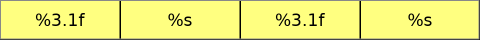
VISUALIZATION VISU_CONFIG_LIGNE_GAZ_SURV_MFC_MKS  // 480x40
VAR_IN_OUT
	m_Input_MASSFLOW:		BLOCK_MFC_MKS_NoCoE;
END_VAR
    Rectangle (0,0 120x40), "%3.1f", text variable: m_Input_MASSFLOW.VAR_ALM_SURV.OFFSET, input disabled if: NOT Global_Variables.PRG_USER.ACTU_USER.CONF_MACHINE
        OnMouseDown: write the text variable via Edit
    Rectangle (240,0 120x40), "%3.1f", text variable: m_Input_MASSFLOW.VAR_DEF_SURV.offset, input disabled if: NOT Global_Variables.PRG_USER.ACTU_USER.CONF_MACHINE
        OnMouseDown: write the text variable via VisuDialogs.Numpad
    Rectangle (120,0 120x40), "%s", text variable: m_Input_MASSFLOW.ALM_SURV.delay, input disabled if: NOT Global_Variables.PRG_USER.ACTU_USER.CONF_MACHINE
        OnMouseDown: write the text variable via VisuDialogs.Keypad
    Rectangle (360,0 120x40), "%s", text variable: m_Input_MASSFLOW.DEF_SURV.DELAY, input disabled if: NOT Global_Variables.PRG_USER.ACTU_USER.CONF_MACHINE
        OnMouseDown: write the text variable via VisuDialogs.Keypad
END_VISUALIZATION

// ---- Visualizations/Symbole/GAZ/VISU_CONFIG_REGUL_GAZ.TcVIS
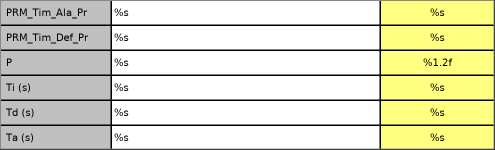
VISUALIZATION VISU_CONFIG_REGUL_GAZ  // 495x150
VAR_IN_OUT
	m_Input_REGULATION : BLOCK_REGUL_PR_GAZ;
END_VAR
    Rectangle (111,50 269x25), "%s", text list: 'TextList_Config_Gaz', text index: 31
    Rectangle (380,50 115x25), "%1.2f", text variable: m_Input_REGULATION.CONTROLEUR_GAZ.CONF_Kp, input disabled if: NOT Global_Variables.PRG_USER.ACTU_USER.CONF_MACHINE
        OnMouseDown: write the text variable via InputWithLimits, min 0
    Rectangle (0,50 111x25), "P", text variable: 1
    Rectangle (111,75 269x25), "%s", text list: 'TextList_Config_Gaz', text index: 32
    Rectangle (111,100 269x25), "%s", text list: 'TextList_Config_Gaz', text index: 33
    Rectangle (380,75 115x25), "%s", text variable: m_Input_REGULATION.CONTROLEUR_GAZ.CONF_Tn, input disabled if: NOT Global_Variables.PRG_USER.ACTU_USER.CONF_MACHINE
        OnMouseDown: write the text variable via InputWithLimits
    Rectangle (0,75 111x25), "Ti (s)", text variable: 1
    Rectangle (380,100 115x25), "%s", text variable: m_Input_REGULATION.CONTROLEUR_GAZ.CONF_Tv, input disabled if: NOT Global_Variables.PRG_USER.ACTU_USER.CONF_MACHINE
        OnMouseDown: write the text variable via InputWithLimits
    Rectangle (0,100 111x25), "Td (s)", text variable: 1
    Rectangle (111,125 269x25), "%s", text list: 'TextList_Config_Gaz', text index: 34
    Rectangle (380,125 115x25), "%s", text variable: m_Input_REGULATION.CONTROLEUR_GAZ.CONF_Td, input disabled if: NOT Global_Variables.PRG_USER.ACTU_USER.CONF_MACHINE
        OnMouseDown: write the text variable via InputWithLimits
    Rectangle (0,125 111x25), "Ta (s)", text variable: 1
    Rectangle (111,0 269x25), "%s", text list: 'TextList_Config_Gaz', text index: 29
    Rectangle (380,0 115x25), "%s", text variable: m_Input_REGULATION.PRM_Tim_Ala_Pr, input disabled if: NOT Global_Variables.PRG_USER.ACTU_USER.CONF_MACHINE
        OnMouseDown: write the text variable via InputWithLimits
    Rectangle (0,0 111x25), "PRM_Tim_Ala_Pr"
    Rectangle (111,25 269x25), "%s", text list: 'TextList_Config_Gaz', text index: 30
    Rectangle (380,25 115x25), "%s", text variable: m_Input_REGULATION.PRM_Tim_Def_Pr, input disabled if: NOT Global_Variables.PRG_USER.ACTU_USER.CONF_MACHINE
        OnMouseDown: write the text variable via InputWithLimits
    Rectangle (0,25 111x25), "PRM_Tim_Def_Pr"
END_VISUALIZATION

// ---- Visualizations/Symbole/GAZ/VISU_LIGNE_GAZ.TcVIS
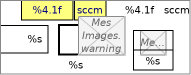
VISUALIZATION VISU_LIGNE_GAZ  // 191x75
VAR_IN_OUT
	m_Input_MACHINE:	BLOCK_MODE_MARCHE_V2_0;
	m_Input_MASSFLOW:	BLOCK_MFC_BROOKS_NoCoE;
	m_Input_LIGNE_GAZ:	BLOCK_LIGNE_GAZ;
END_VAR
    Frame (21,0 170x75)
        shows VISU_MFC_BROOKS(m_Input_MACHINE := m_Input_MACHINE, m_Input_MASSFLOW := m_Input_MASSFLOW, m_Input_LIGNE_GAZ := m_Input_LIGNE_GAZ)
    Frame (133,30 42x42)
        shows VISU_VANNE_2P_H_ACT2(m_Input_VANNE := m_Input_LIGNE_GAZ.VGI)
    Rectangle (0,25 48x28), "%s", text variable: m_Input_MASSFLOW.CONF_Util_Name
END_VISUALIZATION

// ---- Visualizations/Symbole/GAZ/VISU_LIGNE_GAZ_ANA.TcVIS
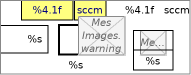
VISUALIZATION VISU_LIGNE_GAZ_ANA  // 191x75
VAR_IN_OUT
	m_Input_MACHINE:	BLOCK_MODE_MARCHE_V2_0;
	m_Input_MASSFLOW:	BLOCK_MFC_ANA2;
	m_Input_LIGNE_GAZ:	BLOCK_LIGNE_GAZ;		
END_VAR
    Frame (21,0 170x75)
        shows VISU_MFC_ANA(m_Input_MACHINE := m_Input_MACHINE, m_Input_MASSFLOW := m_Input_MASSFLOW, m_Input_LIGNE_GAZ := m_Input_LIGNE_GAZ)
    Frame (133,30 42x42)
        shows VISU_VANNE_2P_H_ACT2(m_Input_VANNE := m_Input_LIGNE_GAZ.VGI)
    Rectangle (0,25 48x28), "%s", text variable: m_Input_MASSFLOW.CONF_Util_Name
END_VISUALIZATION

// ---- Visualizations/Symbole/GAZ/VISU_LIGNE_GAZ_VGAUCHE.TcVIS
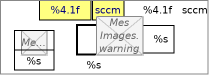
VISUALIZATION VISU_LIGNE_GAZ_VGAUCHE  // 209x75
VAR_IN_OUT
	m_Input_MACHINE:	BLOCK_MODE_MARCHE_V2_0;
	m_Input_MASSFLOW:	BLOCK_MFC_MKS_NoCoE;
	m_Input_LIGNE_GAZ:	BLOCK_LIGNE_GAZ;
END_VAR
    Frame (14,30 42x42)
        shows VISU_VANNE_2P_H_ACT2(m_Input_VANNE := m_Input_LIGNE_GAZ.VGI)
    Rectangle (126,25 48x28), "%s", text variable: m_Input_MASSFLOW.CONF_Util_Name
    Frame (39,0 170x75)
        shows VISU_MFC_MKS(m_Input_MACHINE := m_Input_MACHINE, m_Input_MASSFLOW := m_Input_MASSFLOW, m_Input_LIGNE_GAZ := m_Input_LIGNE_GAZ)
        p3089095539: m_Input_MACHINE
        p1532468285: m_Input_MASSFLOW
        p4266626122: m_Input_LIGNE_GAZ
END_VISUALIZATION

// ---- Visualizations/Symbole/GAZ/VISU_MFC_ANA.TcVIS
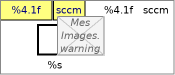
VISUALIZATION VISU_MFC_ANA  // 175x75
VAR_IN_OUT
	m_Input_MACHINE:	BLOCK_MODE_MARCHE_V2_0;
	m_Input_MASSFLOW:	BLOCK_MFC_ANA2;
	m_Input_LIGNE_GAZ:	BLOCK_LIGNE_GAZ;
END_VAR
    Rectangle (37,24 34x31)
    RoundedRectangle (0,0 52x20), "%4.1f", text variable: m_Input_MASSFLOW.PRM_Flow, invisible if: (m_Input_MACHINE.STATE_Manu) <> 0
    Rectangle (90,0 49x20), "%4.1f", text variable: m_Input_MASSFLOW.STATE_Flow
    RoundedRectangle (53,0 32x20), "sccm"
    Rectangle (140,0 35x20), "sccm"
    Rectangle (35,55 40x20), "%s", text variable: m_Input_MASSFLOW.MNEMO
    RoundedRectangle (0,0 52x20), "%4.1f", text variable: m_Input_LIGNE_GAZ.PRM_Flow, invisible if: NOT m_Input_MACHINE.STATE_Manu, input disabled if: NOT m_Input_MACHINE.STATE_Manu OR NOT PRG_User.ACTU_USER.MAINTENANCE
        OnMouseDown: write the text variable via VisuDialogs.Numpad, min 0, max m_Input_MASSFLOW.CONF_Util_Max_Flow
    Polyline (53,32)
    Polyline (61,39)
    Rectangle (55,39 16x18), "D"
    Image (57,16 47x39), invisible if: NOT m_Input_MASSFLOW.STATE_NOK, image: MesImages.warning
END_VISUALIZATION

// ---- Visualizations/Symbole/GAZ/VISU_MFC_BROOKS.TcVIS
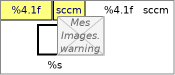
VISUALIZATION VISU_MFC_BROOKS  // 175x75
VAR_IN_OUT
	m_Input_MACHINE:	BLOCK_MODE_MARCHE_V2_0;
	m_Input_MASSFLOW:	BLOCK_MFC_BROOKS_NoCoE;
	m_Input_LIGNE_GAZ:	BLOCK_LIGNE_GAZ;
END_VAR
    Rectangle (37,24 34x31)
    RoundedRectangle (0,0 52x20), "%4.1f", text variable: m_Input_MASSFLOW.PRM_Flow, invisible if: NOT m_Input_MACHINE.STATE_Manu, input disabled if: NOT m_Input_MACHINE.STATE_Manu OR NOT PRG_User.ACTU_USER.MAINTENANCE
    Rectangle (90,0 49x20), "%4.1f", text variable: m_Input_MASSFLOW.STATE_Flow
    RoundedRectangle (53,0 32x20), "sccm"
    Rectangle (140,0 35x20), "sccm"
    Rectangle (35,55 40x20), "%s", text variable: m_Input_MASSFLOW.MNEMO
    RoundedRectangle (0,0 52x20), "%4.1f", text variable: m_Input_LIGNE_GAZ.PRM_Flow, invisible if: NOT m_Input_MACHINE.STATE_Manu, input disabled if: NOT m_Input_MACHINE.STATE_Manu OR NOT PRG_User.ACTU_USER.MAINTENANCE
        OnMouseDown: write the text variable via InputWithLimits, min 0, max m_Input_MASSFLOW.CONF_Util_Max_Flow
    Polyline (53,32)
    Polyline (61,39)
    Rectangle (55,39 16x18), "D"
    Image (57,16 47x39), invisible if: NOT m_Input_MASSFLOW.STATE_NOK, image: MesImages.warning
END_VISUALIZATION

// ---- Visualizations/Symbole/GAZ/VISU_MFC_MKS.TcVIS
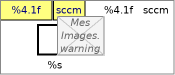
VISUALIZATION VISU_MFC_MKS  // 175x75
VAR_IN_OUT
	m_Input_MACHINE:	BLOCK_MODE_MARCHE_V2_0;
	m_Input_MASSFLOW:	BLOCK_MFC_MKS_NoCoE;
	m_Input_LIGNE_GAZ:	BLOCK_LIGNE_GAZ;
END_VAR
    Rectangle (37,24 34x31)
    RoundedRectangle (0,0 52x20), "%4.1f", text variable: m_Input_MASSFLOW.PRM_Flow, invisible if: (m_Input_MACHINE.STATE_Manu) <> 0
    Rectangle (90,0 49x20), "%4.1f", text variable: m_Input_MASSFLOW.STATE_Flow
    RoundedRectangle (53,0 32x20), "sccm"
    Rectangle (140,0 35x20), "sccm"
    Rectangle (35,55 40x20), "%s", text variable: m_Input_MASSFLOW.MNEMO
    RoundedRectangle (0,0 52x20), "%4.1f", text variable: m_Input_LIGNE_GAZ.PRM_Flow, invisible if: NOT m_Input_MACHINE.STATE_Manu, input disabled if: NOT m_Input_MACHINE.STATE_Manu OR NOT PRG_User.ACTU_USER.MAINTENANCE
        OnMouseDown: write the text variable via VisuDialogs.Numpad, min 0, max m_Input_MASSFLOW.CONF_Util_Max_Flow
    Polyline (53,32)
    Polyline (61,39)
    Rectangle (55,39 16x18), "D"
    Image (57,16 47x39), invisible if: NOT m_Input_MASSFLOW.STATE_NOK, image: MesImages.warning
END_VISUALIZATION

// ---- Visualizations/Symbole/IAD/VISU_MARK3_PLUS.TcVIS
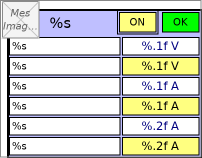
VISUALIZATION VISU_MARK3_PLUS  // 202x158
VAR_IN_OUT
	m_Input_IAD : BLOCK_MARK3_PLUS;
END_VAR
    Rectangle (7,9 195x149)
    Rectangle (162,12 37x20), "NOK", invisible if: (m_Input_IAD.IN_BUSSTAT) <> 0
    Rectangle (119,12 37x20), "OFF", invisible if: (m_Input_IAD.STATE_BEAM OR m_Input_IAD.STATE_BEAM_ON) <> 0
    Rectangle (162,12 37x20), "OK", invisible if: NOT m_Input_IAD.IN_BUSSTAT
    Rectangle (119,12 37x20), "ON", invisible if: NOT m_Input_IAD.STATE_BEAM AND NOT m_Input_IAD.STATE_BEAM_ON
    RoundedRectangle (9,37 111x18), "%s", text list: 'TextList_IAD', text index: 0
    RoundedRectangle (122,37 77x18), "%.1f V", text variable: m_Input_IAD.STATE_V_Anode
    RoundedRectangle (9,77 111x18), "%s", text list: 'TextList_IAD', text index: 1
    RoundedRectangle (122,77 77x18), "%.1f A", text variable: m_Input_IAD.STATE_I_Anode
    Rectangle (119,12 37x20), "ON", invisible if: (m_Input_IAD.STATE_BEAM_ON OR NOT m_Input_IAD.STATE_BEAM) <> 0
    Rectangle (7,12 107x22), "%s", text variable: m_Input_IAD.MNEMO
    Polyline (7,35)
    RoundedRectangle (9,57 111x18), "%s", invisible if: NOT Global_Variables.PRG_USER.ACTU_USER.MAINTENANCE OR NOT MACHINE.State_manu, text list: 'TextList_IAD', text index: 0
    RoundedRectangle (122,57 77x18), "%.1f V", text variable: m_Input_IAD.PRM_ANODE_VOLTAGE, invisible if: NOT Global_Variables.PRG_USER.ACTU_USER.MAINTENANCE OR NOT MACHINE.State_manu
        OnMouseDown: write the text variable via VisuDialogs.Numpad, min 0, max 300
    RoundedRectangle (9,97 111x18), "%s", invisible if: NOT Global_Variables.PRG_USER.ACTU_USER.MAINTENANCE OR NOT MACHINE.State_manu, text list: 'TextList_IAD', text index: 1
    RoundedRectangle (122,97 77x18), "%.1f A", text variable: m_Input_IAD.PRM_ANODE_CURRENT, invisible if: NOT Global_Variables.PRG_USER.ACTU_USER.MAINTENANCE OR NOT MACHINE.State_manu
        OnMouseDown: write the text variable via VisuDialogs.Numpad, min 0, max 15
    Rectangle (117,10 41x24), invisible if: NOT m_Input_IAD.BEAM.AUTOR_ON_IHM AND NOT m_Input_IAD.BEAM.AUTOR_OFF_IHM, input disabled if: ((NOT m_Input_IAD.BEAM.AUTOR_ON_IHM AND NOT m_Input_IAD.BEAM.AUTOR_OFF_IHM) OR NOT PRG_User.ACTU_USER.MAINTENANCE) <> 0
        OnMouseUp: execute { m_Input_IAD.BEAM.M_On:=(TRUE); }
    RoundedRectangle (9,117 111x18), "%s", text list: 'TextList_IAD', text index: 2
    RoundedRectangle (122,117 77x18), "%.2f A", text variable: m_Input_IAD.STATE_I_Neut
    RoundedRectangle (9,137 111x18), "%s", invisible if: NOT Global_Variables.PRG_USER.ACTU_USER.MAINTENANCE OR NOT MACHINE.State_manu, text list: 'TextList_IAD', text index: 2
    RoundedRectangle (122,137 77x18), "%.2f A", text variable: m_Input_IAD.PRM_NEUTRAL_CURRENT, invisible if: NOT Global_Variables.PRG_USER.ACTU_USER.MAINTENANCE OR NOT MACHINE.State_manu
        OnMouseDown: write the text variable via VisuDialogs.Numpad, min 0, max 1.86
    Image (2,1 37x37), invisible if: NOT m_Input_IAD.STATE_Nok, image: MesImages.warning
END_VISUALIZATION

// ---- Visualizations/Symbole/IAD/VISU_MARK3_PLUS_COTE.TcVIS
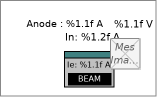
VISUALIZATION VISU_MARK3_PLUS_COTE  // 157x97
VAR_IN_OUT
	m_Input_IAD : BLOCK_MARK3_PLUS;
END_VAR
    Polygon (59,48), invisible if: NOT m_Input_IAD.STATE_BEAM_ON
    Polygon (91,50), invisible if: NOT m_Input_IAD.STATE_BEAM_ON
    Polygon (86,81)
    Rectangle (85,69 25x10), "ON"
    RoundedRectangle (64,51 50x36)
    Rectangle (64,51 50x7)
    RoundedRectangle (68,73 43x12), "BEAM", colour toggle: (m_Input_IAD.STATE_BEAM_ON) <> 0
    Rectangle (51,58 76x14), "Ie: %1.1f A", text variable: m_Input_IAD.STATE_I_Emi, invisible if: NOT m_Input_IAD.STATE_BEAM
    Rectangle (63,52 52x32), input disabled if: ((NOT m_Input_IAD.BEAM.AUTOR_ON_IHM AND NOT m_Input_IAD.BEAM.AUTOR_OFF_IHM) OR NOT PRG_User.ACTU_USER.MAINTENANCE) <> 0
        OnMouseUp: execute { m_Input_IAD.BEAM.M_On:=(TRUE); }
    RoundedRectangle (68,73 43x12), "BEAM", invisible if: (m_Input_IAD.STATE_BEAM_ON OR m_Input_IAD.STATE_BEAM) <> 0
    Rectangle (25,17 83x14), "Anode : %1.1f A", text variable: m_Input_IAD.STATE_I_Anode, invisible if: NOT m_Input_IAD.STATE_BEAM
    Rectangle (107,17 50x14), "%1.1f V", text variable: m_Input_IAD.STATE_V_Anode, invisible if: NOT m_Input_IAD.STATE_BEAM
    Rectangle (60,30 62x14), "In: %1.2f A", text variable: m_Input_IAD.STATE_I_Neut, invisible if: NOT m_Input_IAD.STATE_BEAM
    Polygon (47,55)
    Image (110,38 30x31), invisible if: NOT m_Input_IAD.STATE_Nok, image: MesImages.warning
END_VISUALIZATION

// ---- Visualizations/Symbole/JAUGES/VISU_JAUGE_BCG450_V_HAUT.TcVIS
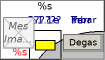
VISUALIZATION VISU_JAUGE_BCG450_V_HAUT  // 105x60
VAR_IN_OUT
	m_Input_JAUGE : BLOCK_BCG450_ANA;
END_VAR
    Rectangle (0,0 105x60), invisible if: TRUE
    Rectangle (0,10 90x20), "??????", invisible if: (m_Input_JAUGE.STATE_OK) <> 0
    Group (31,31 28x28)
        Ellipse (0,0 140x100)
        Rectangle (0,50 140x150)
        Polyline (140,50)
    Rectangle (35,40 20x10), colour toggle: m_Input_JAUGE.OUT_M1, invisible if: m_Input_JAUGE.OUT_DGZ
    Rectangle (10,1 70x10), "%s", text variable: m_Input_JAUGE.MNEMO
    Rectangle (35,40 20x10), invisible if: NOT m_Input_JAUGE.OUT_DGZ
    Rectangle (29,30 32x30), invisible if: NOT (m_Input_JAUGE.Autor_ON_IHM OR m_Input_JAUGE.Autor_Off_IHM ) OR NOT PRG_User.ACTU_USER.MAINTENANCE
        tap m_Input_JAUGE.M_M1
    Group (5,10 88x18), invisible if: NOT m_Input_JAUGE.STATE_OK
        Rectangle (0,0 57x20), "%1.1e", text variable: m_Input_JAUGE.STATE_Pression
        Rectangle (60,0 27x20), "Torr", invisible if: NOT (m_Input_JAUGE.CONF_unit = 1)
        Rectangle (60,0 30x20), "mbar", invisible if: NOT (m_Input_JAUGE.CONF_unit = 0)
        Rectangle (60,0 27x20), "Pa", invisible if: NOT (m_Input_JAUGE.CONF_unit = 2)
    Rectangle (5,47 30x10), "%s", text variable: m_Input_JAUGE.STATE_ERR, invisible if: NOT m_Input_JAUGE.STATE_NOK
    Image (3,17 31x31), invisible if: NOT m_Input_JAUGE.STATE_NOK, image: MesImages.warning
    Button (63,34 40x17), "Degas", invisible if: NOT m_Input_JAUGE.AUTOR_Dgz_IHM OR NOT PRG_User.ACTU_USER.MAINTENANCE
        toggle m_Input_JAUGE.M_DGZ
END_VISUALIZATION

// ---- Visualizations/Symbole/JAUGES/VISU_JAUGE_BCG450_V_HAUT_ETHERCAT.TcVIS
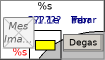
VISUALIZATION VISU_JAUGE_BCG450_V_HAUT_ETHERCAT  // 105x60
VAR_IN_OUT
	m_Input_JAUGE : BLOCK_BCG450_ETHERCAT;
END_VAR
    Rectangle (0,0 105x60), invisible if: TRUE
    Rectangle (0,10 90x20), "??????", invisible if: (m_Input_JAUGE.STATE_OK) <> 0
    Group (31,31 28x28)
        Ellipse (0,0 140x100)
        Rectangle (0,50 140x150)
        Polyline (140,50)
    Rectangle (35,40 20x10), colour toggle: NOT ( m_Input_JAUGE.OP_RAH.Etape.4 OR m_Input_JAUGE.OP_RAH.Etape.5 OR m_Input_JAUGE.OP_RAH.Etape.6 OR m_Input_JAUGE.OP_RAH.Etape.7), invisible if: (m_Input_JAUGE.OP_DGZ.EC) <> 0
    Rectangle (10,1 70x10), "%s", text variable: m_Input_JAUGE.MNEMO
    Rectangle (35,40 20x10), invisible if: NOT m_Input_JAUGE.OP_DGZ.EC
    Rectangle (29,30 32x30), invisible if: NOT (m_Input_JAUGE.Autor_ON_IHM OR m_Input_JAUGE.Autor_Off_IHM ) OR NOT PRG_User.ACTU_USER.MAINTENANCE
        tap m_Input_JAUGE.M_M1
    Group (5,10 88x18), invisible if: NOT m_Input_JAUGE.STATE_OK
        Rectangle (0,0 57x20), "%1.1e", text variable: m_Input_JAUGE.STATE_Pression
        Rectangle (60,0 27x20), "Torr", invisible if: NOT (m_Input_JAUGE.CONF_unit = 1)
        Rectangle (60,0 30x20), "mbar", invisible if: NOT (m_Input_JAUGE.CONF_unit = 0)
        Rectangle (60,0 27x20), "Pa", invisible if: NOT (m_Input_JAUGE.CONF_unit = 2)
    Rectangle (5,47 30x10), "%s", text variable: m_Input_JAUGE.STATE_ERR, invisible if: NOT m_Input_JAUGE.STATE_NOK
    Image (3,17 31x31), invisible if: NOT m_Input_JAUGE.STATE_NOK, image: MesImages.warning
    Button (63,34 40x17), "Degas", invisible if: NOT m_Input_JAUGE.AUTOR_Dgz_IHM OR NOT PRG_User.ACTU_USER.MAINTENANCE
        toggle m_Input_JAUGE.M_DGZ
END_VISUALIZATION

// ---- Visualizations/Symbole/JAUGES/VISU_JAUGE_CDG045_ETHERCAT.TcVIS
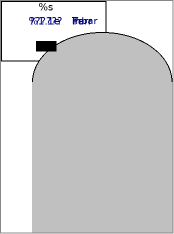
VISUALIZATION VISU_JAUGE_CDG045_ETHERCAT  // 174x234
VAR_IN_OUT
	m_Input_JAUGE:		BLOCK_CDG_ETHERCAT;
END_VAR
    Rectangle (1,1 105x60), invisible if: TRUE
    Rectangle (1,11 90x20), "??????", invisible if: (m_Input_JAUGE.STATE_OK) <> 0
    Group (32,32 28x28)
        Ellipse (0,0 140x100)
        Rectangle (0,50 140x150)
        Polyline (140,50)
    Rectangle (36,41 20x10), colour toggle: TRUE
    Rectangle (11,2 70x10), "%s", text variable: m_Input_JAUGE.MNEMO
    Group (6,11 88x18), invisible if: NOT m_Input_JAUGE.STATE_OK
        Rectangle (0,0 57x20), "%1.1e", text variable: m_Input_JAUGE.STATE_Pression
        Rectangle (60,0 27x20), "Torr", invisible if: NOT (m_Input_JAUGE.CONF_unit = 1)
        Rectangle (60,0 30x20), "mbar", invisible if: NOT (m_Input_JAUGE.CONF_unit = 0)
        Rectangle (60,0 27x20), "Pa", invisible if: NOT (m_Input_JAUGE.CONF_unit = 2)
END_VISUALIZATION

// ---- Visualizations/Symbole/JAUGES/VISU_JAUGE_PCG550_ETHERCAT.TcVIS
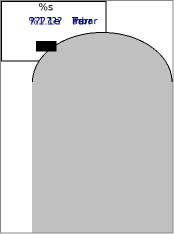
VISUALIZATION VISU_JAUGE_PCG550_ETHERCAT  // 174x234
VAR_IN_OUT
	m_Input_JAUGE:		BLOCK_PCG550_ETHERCAT;
END_VAR
    Rectangle (1,1 105x60), invisible if: TRUE
    Rectangle (1,11 90x20), "??????", invisible if: (m_Input_JAUGE.STATE_OK) <> 0
    Group (32,32 28x28)
        Ellipse (0,0 140x100)
        Rectangle (0,50 140x150)
        Polyline (140,50)
    Rectangle (36,41 20x10), colour toggle: TRUE
    Rectangle (11,2 70x10), "%s", text variable: m_Input_JAUGE.MNEMO
    Group (6,11 88x18), invisible if: NOT m_Input_JAUGE.STATE_OK
        Rectangle (0,0 57x20), "%1.1e", text variable: m_Input_JAUGE.STATE_Pression
        Rectangle (60,0 27x20), "Torr", invisible if: NOT (m_Input_JAUGE.CONF_unit = 1)
        Rectangle (60,0 30x20), "mbar", invisible if: NOT (m_Input_JAUGE.CONF_unit = 0)
        Rectangle (60,0 27x20), "Pa", invisible if: NOT (m_Input_JAUGE.CONF_unit = 2)
END_VISUALIZATION

// ---- Visualizations/Symbole/MESURE/VISU_IC6.TcVIS
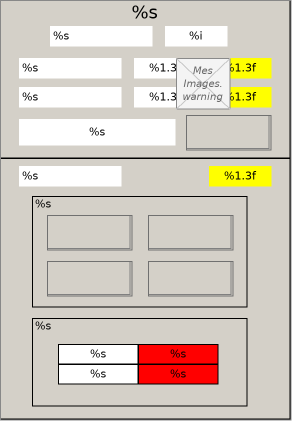
VISUALIZATION VISU_IC6  // 292x421
VAR_IN_OUT
	M_Input_Ctrl:		BLOCK_IC6;
	M_Input_QZ1:		BLOCK_XTAL;
	M_Input_QZ2:		BLOCK_XTAL;
END_VAR
    GroupBox (0,144 290x275), invisible if: NOT M_Input_Ctrl.VISU_Show_Details
        Rectangle (0,14 290x261)
        RoundedRectangle (32,52 215x111), "%s", text list: 'TextList_IC6', text index: 4
        Button (47,71 85x35), input disabled if: NOT PRG_USER.ACTU_USER.MAINTENANCE OR NOT MACHINE.STATE_Manu, text list: 'TextList_IC6', text index: 5
            toggle M_Input_Ctrl.M_Start
        Button (47,117 85x35), text list: 'TextList_IC6', text index: 6
            toggle M_Input_Ctrl.M_Stop
        Button (148,71 85x35), text list: 'TextList_IC6', text index: 7
            toggle M_Input_Ctrl.M_RAZ_Thick
        Button (148,117 85x35), text list: 'TextList_IC6', text index: 8
            toggle M_Input_Ctrl.M_Reset
        Textfield (19,22 102x20), "%s", text list: 'TextList_IC6', text index: 3
        Textfield (209,22 62x20), "%1.3f", text variable: M_Input_Ctrl.STATE_Puissance
        RoundedRectangle (32,174 215x88), "%s", text list: 'TextList_IC6', text index: 9
        Rectangle (58,200 80x20), "%s", text variable: M_Input_QZ1.MNEMO
        Rectangle (58,220 80x20), "%s", text variable: M_Input_QZ2.MNEMO
        Rectangle (138,200 80x20), "OK", invisible if: M_Input_QZ1.STATE_NOK
        Rectangle (138,200 80x20), "%s", invisible if: NOT M_Input_QZ1.STATE_NOK, text list: 'TextList_IC6', text index: 10
        Rectangle (138,220 80x20), "OK", invisible if: M_Input_QZ2.STATE_NOK
        Rectangle (138,220 80x20), "%s", invisible if: NOT M_Input_QZ2.STATE_NOK, text list: 'TextList_IC6', text index: 10
    Rectangle (0,0 290x158), "%s", text variable: M_Input_Ctrl.MNEMO
    Textfield (19,58 102x20), "%s", text list: 'TextList_IC6', text index: 0
    Textfield (19,87 102x20), "%s", text list: 'TextList_IC6', text index: 1
    Textfield (209,58 62x20), "%1.3f", text variable: M_Input_Ctrl.STATE_Global_Rate
    Textfield (209,87 62x20), "%1.3f", text variable: M_Input_Ctrl.STATE_Global_Thick
    Textfield (134,58 62x20), "%1.3f", text variable: M_Input_Ctrl.I_Rate_App
    Textfield (134,87 62x20), "%1.3f", text variable: M_Input_Ctrl.I_Epaisseur
    RoundedRectangle (19,119 156x26), "%s", text variable: M_Input_Ctrl.STATE_Phase
    Image (176,58 54x51), invisible if: NOT M_Input_Ctrl.STATE_NOK, image: MesImages.warning
    Button (186,115 85x35), text list: 'TextList_IC6', text index: 2
        toggle M_Input_Ctrl.VISU_Show_Details
    Textfield (50,26 102x20), "%s", text list: 'TextList_IC6', text index: 11
    Textfield (165,26 62x20), "%i", text variable: M_Input_Ctrl.PRM_Materiau, input disabled if: MACHINE.STATE_Prod
        OnMouseClick: write the text variable via Default, min 1, max 6
END_VISUALIZATION

// ---- Visualizations/Symbole/MESURE/VISU_XTC.TcVIS
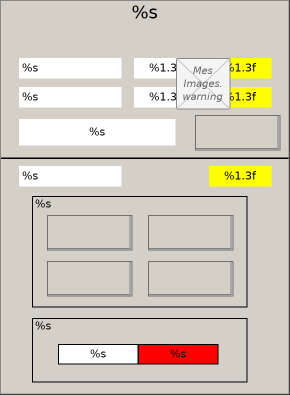
VISUALIZATION VISU_XTC  // 290x395
VAR_IN_OUT
	M_Input_Evap:		BLOCK_EVAP;
	M_Input_Ctrl:		BLOCK_XTC3;
	M_Input_QZ1:		BLOCK_XTAL6;
END_VAR
    GroupBox (0,144 290x251), invisible if: NOT M_Input_Ctrl.VISU_Show_Details
        Rectangle (0,14 290x237)
        RoundedRectangle (32,52 215x111), "%s", text list: 'TextList_IC6', text index: 4
        Button (47,71 85x35), input disabled if: NOT PRG_USER.ACTU_USER.MAINTENANCE OR NOT MACHINE.STATE_Manu, text list: 'TextList_IC6', text index: 5
            toggle M_Input_Ctrl.M_Start
        Button (47,117 85x35), input disabled if: NOT PRG_USER.ACTU_USER.MAINTENANCE OR NOT MACHINE.STATE_Manu, text list: 'TextList_IC6', text index: 6
            toggle M_Input_Ctrl.M_Stop
        Button (148,71 85x35), input disabled if: NOT PRG_USER.ACTU_USER.MAINTENANCE OR NOT MACHINE.STATE_Manu, text list: 'TextList_IC6', text index: 7
            toggle M_Input_Ctrl.M_RAZ_Thick
        Button (148,117 85x35), input disabled if: NOT PRG_USER.ACTU_USER.MAINTENANCE OR NOT MACHINE.STATE_Manu, text list: 'TextList_IC6', text index: 8
            toggle M_Input_Ctrl.M_Reset
        Textfield (19,22 102x20), "%s", text list: 'TextList_IC6', text index: 3
        Textfield (209,22 62x20), "%1.3f", text variable: M_Input_Ctrl.STATE_Power
        RoundedRectangle (32,174 215x64), "%s", text list: 'TextList_IC6', text index: 9
        Rectangle (58,200 80x20), "%s", text variable: M_Input_QZ1.MNEMO
        Rectangle (138,200 80x20), "OK", invisible if: M_Input_QZ1.STATE_NOK
        Rectangle (138,200 80x20), "%s", invisible if: NOT M_Input_QZ1.STATE_NOK, text list: 'TextList_IC6', text index: 10
    Rectangle (0,0 290x158), "%s", text variable: M_Input_Ctrl.MNEMO
    Textfield (19,58 102x20), "%s", text list: 'TextList_IC6', text index: 0
    Textfield (19,87 102x20), "%s", text list: 'TextList_IC6', text index: 1
    Textfield (209,58 62x20), "%1.3f", text variable: M_Input_Ctrl.STATE_Rate
    Textfield (209,87 62x20), "%1.3f", text variable: M_Input_Ctrl.STATE_Thickness
    Textfield (134,58 62x20), "%1.3f", text variable: M_Input_Evap.PRM_Rate, input disabled if: NOT Global_Variables.PRG_USER.ACTU_USER.MAINTENANCE OR NOT MACHINE.STATE_Manu
    Textfield (134,87 62x20), "%1.3f", text variable: M_Input_Evap.PRM_Thickness, input disabled if: NOT Global_Variables.PRG_USER.ACTU_USER.MAINTENANCE OR NOT MACHINE.STATE_Manu
    RoundedRectangle (19,119 156x26), "%s", text variable: M_Input_Ctrl.STATE_Phase
    Image (176,58 54x51), invisible if: NOT M_Input_Ctrl.STATE_NOK, image: MesImages.warning
    Button (195,115 85x35), text list: 'TextList_IC6', text index: 2
        toggle M_Input_Ctrl.VISU_Show_Details
END_VISUALIZATION

// ---- Visualizations/Symbole/MODE_MARCHE/VISU_BANDEAU.TcVIS
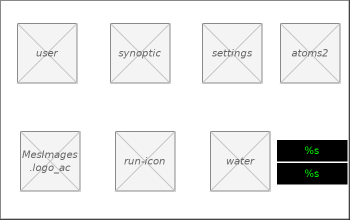
VISUALIZATION VISU_BANDEAU  // 350x220
VAR_INPUT
	m_Input_MACHINE : BLOCK_MODE_MARCHE_V2_0;
END_VAR
    Rectangle (0,0 350x220)
    Image (115,131 60x60), image: run-icon
        toggle Global_Variables.SHOW_SM_SA
        OnMouseClick: change screen: VISU_SA
    Image (202,23 60x60), image: settings
        OnMouseClick: execute { Global_Variables.SHOW_SM_SA:=(FALSE); }
        OnMouseClick: change screen: VISU_CONFIG_POMPAGE
    Image (17,23 60x60), image: user
        OnMouseClick: execute { Global_Variables.SHOW_SM_SA:=(FALSE); }
        OnMouseClick: change screen: UTIL_MENU
    Image (20,131 60x60), image: MesImages.logo_ac
        OnMouseClick: execute { Global_Variables.SHOW_SM_SA:=(FALSE); }
        OnMouseClick: change screen: SYN_INFOS
    Image (110,23 60x60), image: synoptic
        OnMouseClick: execute { Global_Variables.SHOW_SM_SA:=(FALSE); }
        OnMouseClick: change screen: SYN_PROC
    Image (210,131 60x60), image: water
        OnMouseClick: execute { Global_Variables.SHOW_SM_SA:=(FALSE); }
        OnMouseClick: change screen: SYN_SERVITUDES
    Image (280,23 60x60), image: atoms2
        OnMouseClick: execute { Global_Variables.SHOW_SM_SA:=(FALSE); }
        OnMouseClick: change screen: SYN_EXEC_PROC
    Rectangle (277,163 70x21), "%s", text variable: PRG_SEC.STATE_Time
    Rectangle (277,140 70x21), "%s", text variable: PRG_SEC.STATE_Date
END_VISUALIZATION

// ---- Visualizations/Symbole/MODE_MARCHE/VISU_BLANCK_MANUEL.TcVIS
VISUALIZATION VISU_BLANCK_MANUEL  // 1280x1024
END_VISUALIZATION

// ---- Visualizations/Symbole/MODE_MARCHE/VISU_ECOMODE.TcVIS
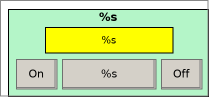
VISUALIZATION VISU_ECOMODE  // 209x97
    RoundedRectangle (8,9 201x88), "%s", text list: 'TextList_EcoMode', text index: 8
    RoundedRectangle (45,27 128x26), "%s", invisible if: NOT MACHINE.STATE_Standby, text list: 'TextList_EcoMode', text index: 10
    Button (62,59 94x30), "%s", text list: 'TextList_EcoMode', text index: 9
        OnMouseClick: change screen: VISU_CONFIG_ECOMODE
    Button (16,59 41x30), "On", invisible if: MACHINE.STATE_Standby, input disabled if: MACHINE.STATE_Prod
        toggle MACHINE.M_Standby
    Button (161,59 41x30), "Off", invisible if: NOT MACHINE.STATE_Standby, input disabled if: MACHINE.STATE_Prod
        toggle MACHINE.M_End_Standby
END_VISUALIZATION

// ---- Visualizations/Symbole/MODE_MARCHE/VISU_ECOMODE_EVAP.TcVIS
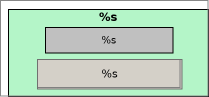
VISUALIZATION VISU_ECOMODE_EVAP  // 209x97
    RoundedRectangle (8,9 201x88), "%s", text list: 'TextList_EcoMode', text index: 8
    RoundedRectangle (45,27 128x26), "%s", colour toggle: PRG_EVAP.VISU_STOP_ECO_MANU, text list: 'TextList_EcoMode', text index: 10
    Button (37,59 145x30), "%s", text list: 'TextList_EcoMode', text index: 6
        toggle PRG_EVAP.VISU_STOP_ECO_MANU
END_VISUALIZATION

// ---- Visualizations/Symbole/MODE_MARCHE/VISU_EV_EXTRAIT.TcVIS
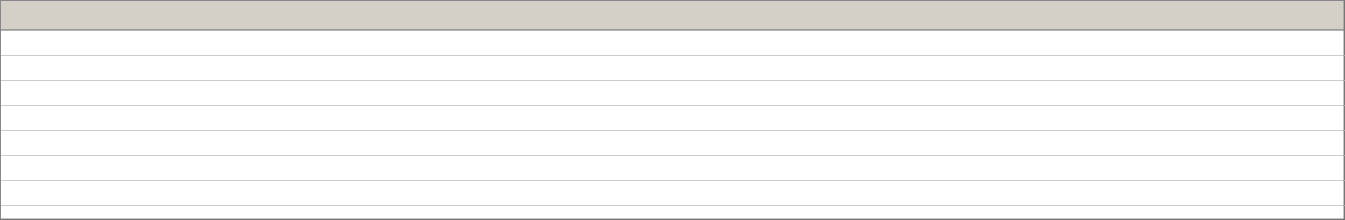
VISUALIZATION VISU_EV_EXTRAIT  // 1345x220
    Table (0,0 1345x220), data array: PRG_DEF_MANAGEMENT.EVENT_LIST
        p2232123230: PRG_DEF_MANAGEMENT.EVENT_LIST[INDEX].STATE_dt
        p511219082: PRG_DEF_MANAGEMENT.EVENT_LIST[INDEX].STATE_App
        p1755163831: PRG_DEF_MANAGEMENT.EVENT_LIST[INDEX].STATE_Path
        p4092479075: PRG_DEF_MANAGEMENT.EVENT_LIST[INDEX].STATE_Title
END_VISUALIZATION

// ---- Visualizations/Symbole/MODE_MARCHE/VISU_FCTS_SA.TcVIS
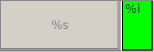
VISUALIZATION VISU_FCTS_SA  // 154x52
VAR_INPUT
	m_Input_ID_XML: UDINT;
END_VAR
VAR_IN_OUT
	m_Input_Operation:	BLOCK_OPERATION;
END_VAR
VAR_INPUT
	m_Input_UserRight:	BOOL;
END_VAR
    Button (0,0 120x50), "%s", invisible if: NOT m_Input_Operation.AUTOR_IHM OR NOT m_Input_UserRight, text list: 'TextList_SA_Operations', text index: m_Input_ID_XML
        toggle m_Input_Operation.ON_IHM
    RoundedRectangle (122,0 30x50), "%i", text variable: m_Input_Operation.STATUS, invisible if: NOT m_Input_Operation.AR
    Button (0,0 120x50), "%s", invisible if: m_Input_Operation.AUTOR_IHM AND m_Input_UserRight, text list: 'TextList_SA_Operations', text index: m_Input_ID_XML
    RoundedRectangle (122,0 30x50), "%i", text variable: m_Input_Operation.STATUS, invisible if: NOT m_Input_Operation.EC
    RoundedRectangle (122,0 30x50), "%i", text variable: m_Input_Operation.STATUS, invisible if: NOT m_Input_Operation.OK
END_VISUALIZATION

// ---- Visualizations/Symbole/MODE_MARCHE/VISU_MODE_MARCHE.TcVIS
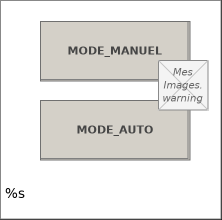
VISUALIZATION VISU_MODE_MARCHE  // 222x220
VAR_IN_OUT
	m_Input_MACHINE : BLOCK_MODE_MARCHE_V2_0;
END_VAR
    Rectangle (0,0 222x220)
    Rectangle (2,170 219x47), "%s", text list: 'TextList_STATE_Mode_Marche', text index: m_Input_MACHINE.STATUS
    Button (40,21 150x60), "MODE_MANUEL", colour toggle: m_Input_MACHINE.STATE_Manu, input disabled if: NOT m_Input_MACHINE.AUTOR_Manu_Ihm OR PRG_SEC.VERROU OR NOT PRG_USER.ACTU_USER.MAINTENANCE
        OnMouseClick: toggle m_Input_MACHINE.M_Manu
    Button (40,100 150x60), "MODE_AUTO", colour toggle: m_Input_MACHINE.STATE_Auto, input disabled if: NOT m_Input_MACHINE.AUTOR_Auto_Ihm
        OnMouseClick: toggle m_Input_MACHINE.M_Auto
    Image (158,60 50x50), invisible if: .STATE_Charg_Persistentes_Ok, image: MesImages.warning
END_VISUALIZATION

// ---- Visualizations/Symbole/MOUVEMENTS PS/AXE STD1/FCT_Part/VISU_AXE_STD1_FCT_MANU.TcVIS
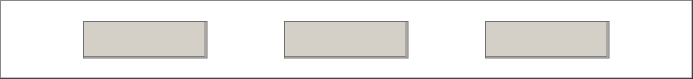
VISUALIZATION VISU_AXE_STD1_FCT_MANU  // 693x79
VAR_IN_OUT
	m_Input_MOTEUR: BLOCK_AXE_STD1;
	m_Input_PRG_MOUVEMENT_PS: BLOCK_PRG_MOUVEMENT_PS;
END_VAR
VAR_INPUT
	m_Input_INDEX_MOTEUR : INT;
END_VAR
    Rectangle (0,0 693x79)
    Button (83,21 124x37), invisible if: NOT .PRG_USER.ACTU_USER.MAINTENANCE OR NOT m_Input_MOTEUR.MANUAL, text list: 'TextList_Moteurs', text index: 0
        tap m_Input_MOTEUR.CO_RESET
    Button (284,21 124x37), invisible if: NOT PRG_USER.ACTU_USER.MAINTENANCE OR NOT m_Input_MOTEUR.MANUAL OR NOT m_Input_MOTEUR.CONF_No_Ref, input disabled if: NOT m_Input_MOTEUR.OP_Validation.AR, text list: 'TextList_Moteurs', text index: 1
        tap m_Input_MOTEUR.M_BIAS
    Button (485,21 124x37), invisible if: NOT PRG_USER.ACTU_USER.MAINTENANCE OR NOT m_Input_MOTEUR.MANUAL OR NOT m_Input_PRG_MOUVEMENT_PS.CONF_Jog[m_Input_INDEX_MOTEUR], text list: 'TextList_Moteurs', text index: 2
        tap m_Input_MOTEUR.CO_Devalid
END_VISUALIZATION

// ---- Visualizations/Symbole/MOUVEMENTS PS/AXE STD1/FCT_Part/VISU_AXE_STD1_FCT_MANU_OSC.TcVIS
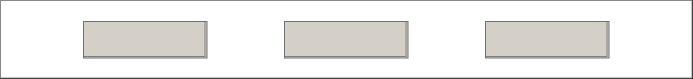
VISUALIZATION VISU_AXE_STD1_FCT_MANU_OSC  // 693x79
VAR_IN_OUT
	m_Input_MOTEUR: BLOCK_AXE_STD1_OSCILLANT;
	m_Input_PRG_MOUVEMENT_PS: BLOCK_PRG_MOUVEMENT_PS;
END_VAR
VAR_INPUT
	m_Input_INDEX_MOTEUR : INT;
END_VAR
    Rectangle (0,0 693x79)
    Button (83,21 124x37), invisible if: NOT .PRG_USER.ACTU_USER.MAINTENANCE OR NOT m_Input_MOTEUR.MANUAL, text list: 'TextList_Moteurs', text index: 0
        tap m_Input_MOTEUR.CO_RESET
    Button (284,21 124x37), invisible if: NOT PRG_USER.ACTU_USER.MAINTENANCE OR NOT m_Input_MOTEUR.MANUAL OR NOT m_Input_MOTEUR.CONF_No_Ref, input disabled if: NOT m_Input_MOTEUR.OP_Validation.AR, text list: 'TextList_Moteurs', text index: 1
        tap m_Input_MOTEUR.AXE_SetPosOffset.Execute
    Button (485,21 124x37), invisible if: NOT PRG_USER.ACTU_USER.MAINTENANCE OR NOT m_Input_MOTEUR.MANUAL OR NOT m_Input_PRG_MOUVEMENT_PS.CONF_Jog[m_Input_INDEX_MOTEUR], text list: 'TextList_Moteurs', text index: 2
        tap m_Input_MOTEUR.CO_Devalid
END_VISUALIZATION

// ---- Visualizations/Symbole/MOUVEMENTS PS/AXE STD1/FCT_Part/VISU_AXE_STD1_FCT_OP.TcVIS
